TEXTLIST AxesConfigTextList
  0 = 'General'
  1 = 'Known positions'
  2 = 'Location'
  3 = 'Local conditions'
  4 = 'AZI axis (1)'
  5 = 'AZI axis (2)'
  6 = 'AZI axis (3)'
  7 = 'ELE axis (1)'
  8 = 'ELE axis (2)'
  9 = 'ROC axis (1)'
  10 = 'ROC axis (2)'
  11 = 'RON axis (1)'
  12 = 'RON axis (2)'
  13 = 'FW axis'
   = ''
END_TEXTLIST

(* stored: Version 1.1.0.1, ProductVersion 3.1.4019.2
   TextList AxesConfigTextList: Id {40b35474-5a5e-41b8-a729-21fcb5517615} *)
